(* CoDeSys 2.3.6.0 project: KOKEV_G53RT_8.pro *)
(* Libraries: STANDARD.LIB 5.6.98 12:03:02 *)

(* Task configuration *)
TASK Standard (PRIORITY := 0, INTERVAL := T#4ms);
	Nockenschaltwerk();
END_TASK

(* Global variable list: Globale_Variablen *)
VAR_GLOBAL
	E1  AT %IX0.0 : BOOL; (* Eingang 1 *)
	E2  AT %IX0.1 : BOOL; (* Eingang 2 *)
	E3  AT %IX0.2 : BOOL; (* Eingang 3 *)
	E4  AT %IX0.3 : BOOL; (* Eingang 4 *)
	E5  AT %IX0.4 : BOOL; (* Eingang 5 *)
	E6  AT %IX0.5 : BOOL; (* Eingang 6 *)
	E7  AT %IX0.6 : BOOL; (* Eingang 7 *)
	E8  AT %IX0.7 : BOOL; (* Eingang 8 *)

       E9  AT %IX1.0 : BOOL; (* Eingang 9 *)
	E10  AT %IX1.1 : BOOL; (* Eingang 10 *)
	E11  AT %IX1.2 : BOOL; (* Eingang 11 *)
	E12  AT %IX1.3 : BOOL; (* Eingang 12 *)
	E13  AT %IX1.4 : BOOL; (* Eingang 13 *)
	E14  AT %IX1.5 : BOOL; (* Eingang 14 *)
	_KS1_UmlRolleGeschl  AT %IX1.6 : BOOL; (* Speicher 1 ist geschloßen *)
	_KS2_UmlRolleGeschl  AT %IX1.7 : BOOL; (* Speicher 2 ist geschloßen *)

	E17  AT %IX2.0 : BOOL; (* Eingang 17 *)
	E18  AT %IX2.1 : BOOL; (* Eingang 18 *)
	E19  AT %IX2.2 : BOOL; (* Eingang 19 *)
	E20  AT %IX2.3 : BOOL; (* Eingang 20 *)
	E21  AT %IX2.4 : BOOL; (* Eingang 21 *)
	E22  AT %IX2.5 : BOOL; (* Eingang 22 *)
	E23  AT %IX2.6 : BOOL; (* Eingang 23 *)
	E24  AT %IX2.7 : BOOL; (* Eingang 24 *)

	T_Quitt_NA  AT %IX3.0 : BOOL; (* Eingang 9 *)
	T_Qiutt_Stoerung  AT %IX3.1 : BOOL; (* Eingang 10 *)
	T_Hand  AT %IX3.2 : BOOL; (* Eingang 11 *)
	T_Auto  AT %IX3.3 : BOOL; (* Eingang 12 *)
	T_Visu  AT %IX3.4 : BOOL; (* Eingang 13 *)
	T_KammBild  AT %IX3.5 : BOOL; (* Eingang 14 *)
	T_Start  AT %IX3.6 : BOOL; (* Eingang 15 *)
	T_Stop  AT %IX3.7 : BOOL; (* Eingang 16 *)

	ET9   AT %IX4.0 : BOOL; (* Eingang 17 *)
	ET10  AT %IX4.1 : BOOL; (* Eingang 18 *)
	ET11  AT %IX4.2 : BOOL; (* Eingang 19 *)
	ET12  AT %IX4.3 : BOOL; (* Eingang 20 *)
	ET13  AT %IX4.4 : BOOL; (* Eingang 21 *)
	ET14  AT %IX4.5 : BOOL; (* Eingang 22 *)
	T_KettenAnfang  AT %IX4.6 : BOOL; (* Eingang 23 *)
	ET16  AT %IX4.7 : BOOL; (* Eingang 24 *)


	IA_Pos_KS1_Input  AT%IW8:INT;	 	(*Speicher 1 Füllstand analoger Eingang*)
	IA_Pos_KS2_Input	AT%IW12:INT;   	(*Speicher 2 Füllstand analoger Eingang*)
	VW_Act_Pos_KS1: INT;					(*Aktueller Füllstand Kettenspeicher 1 skaliert*)
	VW_Act_Pos_KS2:INT;					(*Aktueller Füllstand Kettenspeicher 2 skaliert*)
	IA_EW3	AT%IW12:INT; 				(*Analogeingang 3*)
	IA_EW4  	AT%IW16:INT; 				(*Analogeingang 4*)
	IC_SSI_DG_Input  AT %ID20:UDINT;	(* Drehgeber *)
	My_IC_SSI_DG_Input:UDINT;

	_PneumPressEin  AT %QX0.0 : BOOL; (* Ventil Pneumatik  *)
	A2  AT %QX0.1 : BOOL; (* Ausgang 2 *)
	A3  AT %QX0.2 : BOOL; (* Ausgang 3 *)
	A4  AT %QX0.3 : BOOL; (* Ausgang 4 *)
	A5  AT %QX0.4 : BOOL; (* Ausgang 5 *)
	A6  AT %QX0.5 : BOOL; (* Ausgang 6 *)
	A7  AT %QX0.6 : BOOL; (* Ausgang 7 *)
	A8  AT %QX0.7 : BOOL; (* Ausgang 8 *)

	Q_KS2_EnOutput  AT %QX1.0 : BOOL; (* Ausgang 9 *)
	A10  AT %QX1.1 : BOOL; (* Ausgang 10 *)
	A11  AT %QX1.2 : BOOL; (* Ausgang 11 *)
	A12  AT %QX1.3 : BOOL; (* Ausgang 12 *)
	A13  AT %QX1.4 : BOOL; (* Ausgang 13 *)
	A14  AT %QX1.5 : BOOL; (* Ausgang 14 *)
	A15  AT %QX1.6 : BOOL; (* Ausgang 15 *)
	A16  AT %QX1.7 : BOOL; (* Ausgang 16 *)

	H_Quitt_NA  AT %QX2.0 : BOOL; (* Ausgang 1 *)
	H_Quitt_Stoerung  AT %QX2.1 : BOOL; (* Ausgang 2 *)
	H_Hand  AT %QX2.2 : BOOL; (* Ausgang 3 *)
	H_Auto  AT %QX2.3 : BOOL; (* Ausgang 4 *)
	H_Visu  AT %QX2.4 : BOOL; (* Ausgang 5 *)
	H_KammBild  AT %QX2.5 : BOOL; (* Ausgang 6 *)
	H_Start  AT %QX2.6 : BOOL; (* Ausgang 7 *)
	H_Stop  AT %QX2.7 : BOOL; (* Ausgang 8 *)

	AT9  AT %QX3.0 : BOOL; (* Ausgang 9 *)
	AT10  AT %QX3.1 : BOOL; (* Ausgang 10 *)
	AT11  AT %QX3.2 : BOOL; (* Ausgang 11 *)
	AT12  AT %QX3.3 : BOOL; (* Ausgang 12 *)
	AT13  AT %QX3.4 : BOOL; (* Ausgang 13 *)
	AT14  AT %QX3.5 : BOOL; (* Ausgang 14 *)
	H_KettenAnfang  AT %QX3.6 : BOOL; (* Ausgang 15 *)
	AT16  AT %QX3.7 : BOOL; (* Ausgang 16 *)


	QA_Sollw_Mot1   AT%QW4:WORD; (*Ausgangswort 1*)
	QA_Sollw_Mot2   AT%QW8:WORD; (*Ausgangswort 2*)

	KettenTypen			AT%QW100:ARRAY [1..10,0..10] OF INT ;	(* Es können maximal 10 Kettentypen definiert und remanent gespeichert werden *)
	AKT_KettenTyp		AT%QW420:INT;								(* Nummer des gültigen Kettentyps ( 1-10)   *)
	Speicher_Reg: ARRAY[0..500] OF WORD;							(* Speicherregister für Glieder es werden maximal 500 Glieder beobachtet *)
	Ketten_Reg: ARRAY[0..220] OF WORD;								(* Kettenregister für dien Aktuellen Kettentyp *)
	Z_AKT_KettenTyp_Max:INT;											(* Länge des Aktuellen Kettentyps *)
	Zeiger_Speicher_Trennstelle: INT;									(* Zeiger für die Glieder in der Anlage zeigt auf das Glied unter der Trennstelle *)
	Zeiger_Kette_Trennstelle:INT;										(* Zeiger für die Glieder der Kette zeigt auf das Glied unter der Trennstelle*)
	Zeiger_Loeschen: INT;												(* Zeiger zum Löschen der Register beim Überlauf *)
	M1:BOOL;

	CTU1: CTU;
END_VAR

(* Data type *)
TYPE DriveControl :
STRUCT
	ManOn: BOOL := FALSE; (* Visu -> SPS: Antrieb ein (nur bei FU-Antrieben) *)
	ManOff: BOOL := FALSE; (* Visu -> SPS: Antrieb aus (nur bei FU-Antrieben) *)
	ManFwd: BOOL := FALSE; (* Visu -> SPS: Antrieb im Handbetrieb langsam vorwärts *)
	ManBwd: BOOL := FALSE; (* Visu -> SPS: Antrieb im Handbetrieb langsam rückwärts *)
	TeilungVor: BOOL := FALSE; (* Visu -> SPS: Kette um eine Teilung vor (nur bei Servo-Antrieben) *)
	TeilungZur: BOOL := FALSE; (* Visu -> SPS: Kette um eine Teilung zurück (nur bei Servo-Antrieben) *)
	EnManCtrl: BOOL := FALSE; (* SPS -> Visu: Freigabe manuelle Steuerung *)
	ActOn: BOOL := FALSE; (* SPS -> Visu: Antrieb eingeschaltet *)
	ActOff: BOOL := FALSE; (* SPS -> Visu: Antrieb ausgeschaltet *)
	Error: BOOL := FALSE; (* SPS -> Visu: Störung Antrieb *)
END_STRUCT
END_TYPE

(* Data type *)
TYPE KettenTyp :
STRUCT
	PF: ARRAY [0..19] OF UDINT := 0,410,819,1229,1638,2048,2458,2867,3277,3686,4049,4506,4915,5328,5734,6144,6554,6963,7373,7782;

END_STRUCT
END_TYPE

(* Data type *)
TYPE KS_Control :
STRUCT
	EnInput: BOOL := FALSE; (* Freigabe Befüllen *)
	EnOutput: BOOL := FALSE; (* Freigabe Entleeren *)
	ActState: INT := 0; (* aktueller zustand für Visu *)
END_STRUCT
END_TYPE

(* Data type *)
TYPE MotorControl :
STRUCT
	ManOn: BOOL := FALSE; (* Visu -> SPS: Antrieb im Handbetrieb ein *)
	ManOff: BOOL := FALSE; (* Visu -> SPS: Antrieb im Handbetrieb aus *)
	EnManCtrl: BOOL := FALSE; (* SPS -> Visu: Freigabe manuelle Steuerung *)
	ActOn: BOOL := FALSE; (* SPS -> Visu: Antrieb eingeschaltet *)
	ActOff: BOOL := FALSE; (* SPS -> Visu: Antrieb ausgeschaltet *)
	Error: BOOL := FALSE; (* SPS -> Visu: Störung Antrieb *)
END_STRUCT
END_TYPE

(* Data type *)
TYPE PneumControl :
STRUCT
	SetOn: BOOL := FALSE; (* Visu -> SPS: Arbeitsstellung anfahren *)
	SetOff: BOOL := FALSE; (* Visu -> SPS: Grundstellung anfahren *)
	EnSet: BOOL := FALSE; (* SPS -> Visu: Freigabe manuell Steuerung *)
	ActOn: BOOL := FALSE; (* SPS -> Visu: Zylinder in Arbeitsstellung *)
	ActOff: BOOL := FALSE; (* SPS -> Visu: Zylinder in Grundstellung *)
	Error: BOOL := FALSE; (* SPS -> Visu: Störung Zylinder oder Endschalter *)
END_STRUCT
END_TYPE

(* Data type *)
TYPE PosControl :
STRUCT
	PosSet: INT := 0; (* Positionssollwert [mm] *)
	ActPos: INT := 0; (* Positionsistwert [mm] *)
	PosLimitLo: INT := 0; (* unterer Grenzwert Sollposition [mm] *)
	PosLimitHi: INT := 0; (* oberer Grenzwert Sollposition [mm] *)
	StartPos: BOOL := FALSE; (* Visu -> SPS: Positionierung starten *)
	StoppPos: BOOL := FALSE; (* Visu -> SPS: Positionierung abbrechen *)
	ManPosUp: BOOL := FALSE; (* Visu -> SPS: Handbetrieb Positon erhöhen *)
	ManPosDn: BOOL := FALSE; (* Visu -> SPS: Handbetrieb Positon verringern *)
	EnPosSet: BOOL := FALSE; (* SPS -> Visu: Freigabe Sollwerteingabe *)
	EnManPos: BOOL := FALSE; (* SPS -> Visu: Freigabe manuelle Positionierung *)
	ActOn: BOOL := FALSE; (* SPS -> Visu: Antrieb eingeschaltet *)
	ActOff: BOOL := FALSE; (* SPS -> Visu: Antrieb ausgeschaltet *)
	Error: BOOL := FALSE; (* SPS -> Visu: Störung Antrieb *)
END_STRUCT
END_TYPE

(* Data type *)
TYPE StationControl :
STRUCT
	StepCounter: INT; (* SPS -> Visu: Schrittzähler *)
	SingleStep: BOOL := FALSE; (* Visu -> SPS: Einzelschritt weiterschalten *)
	SingleCycle: BOOL := FALSE; (* Visu -> SPS: Einzelzyklus ausführen *)
	StartCycle: BOOL := FALSE; (* Zyklus im Auto-Betrieb starten *)
	ManInit: BOOL := FALSE; (* Visu -> SPS: Grundstellung anfahren *)
	AutoInit: BOOL := FALSE; (* Grundstellung im Auto-Betrieb anfahren *)
	SetFinished: BOOL := FALSE; (* Visu -> SPS: Fertigmeldung setzen *)
	WaitPos: BOOL := FALSE; (* Station in Warteposition für Stopp *)
	EnSemiAutoCtrl: BOOL := FALSE; (* SPS -> Visu: Steuerung Halbautomatikbetrieb freigeben; Freigabe für SingleStep, SingleCycle, InitPos und SetFinished *)
	InitPos: BOOL := FALSE; (* Station in Grundstellung *)
	Finished: BOOL := FALSE; (* Station fertig *)
	ErrorInitPos: BOOL := FALSE; (* Störung Grundstellung nicht erreicht *)
	ErrorCycleTime: BOOL := FALSE; (* Störung Zeitüberschreitung Zyklus *)
	ActState: INT := 0; (* SPS -> Visu: Zustand der Station: 0 = Störung, 1 = bereit, 2 = aktiv *)
END_STRUCT
END_TYPE

(* POU Nockenschaltwerk, ST *)
PROGRAM Nockenschaltwerk
VAR
	Zeiger :INT:=0;
	Nocke:BOOL:=FALSE;
	Zaeler:WORD;
	Skal_IC_SSI_DG_Input: DINT;
	Skal_IC_SSI_DG_Input_Alt:DINT;
	Skal_IC_SSI_DG_Input_Delta:DINT;
	CTU2:WORD;
END_VAR
(*  Miroslav Knezevic TCM 19.03.07  *)
(*  Das Nockenschaltwerk liefert 20 Impulse bei einer Umdrehung des SSI Drehgebers *)
(* Voller Kreis = 8192 Inkremente,  1 Impuls= 20 Inkremente *)



Skal_IC_SSI_DG_Input:=IC_SSI_DG_Input* 20 / 256;
Skal_IC_SSI_DG_Input_Delta:=Skal_IC_SSI_DG_Input - Skal_IC_SSI_DG_Input_Alt;

IF Skal_IC_SSI_DG_Input_Delta<-5 THEN
	Skal_IC_SSI_DG_Input_Delta:=1;
END_IF

IF Skal_IC_SSI_DG_Input_Delta>5 THEN
	Skal_IC_SSI_DG_Input_Delta:=-1;
END_IF

Zeiger_Speicher_Trennstelle:=DINT_TO_INT(Zeiger_Speicher_Trennstelle+Skal_IC_SSI_DG_Input_Delta);
IF Zeiger_Speicher_Trennstelle>500 THEN
	Zeiger_Speicher_Trennstelle:=1;
END_IF
IF Zeiger_Speicher_Trennstelle<1 THEN
	Zeiger_Speicher_Trennstelle:=500;
END_IF

CTU1(
	CU:=M1 ,
	RESET:= ,
	PV:=500 ,
	Q=> ,
	CV=> );

CTU2:=CTU1.CV;


Zeiger_Kette_Trennstelle:=DINT_TO_INT(Zeiger_Kette_Trennstelle+Skal_IC_SSI_DG_Input_Delta);
IF Zeiger_Kette_Trennstelle>Z_AKT_KettenTyp_Max THEN
	Zeiger_Kette_Trennstelle:=1;
END_IF

IF Zeiger_Kette_Trennstelle<1 THEN
	Zeiger_Kette_Trennstelle:=Z_AKT_KettenTyp_Max;
END_IF

IF ABS(Skal_IC_SSI_DG_Input_Delta)>1 THEN
		M1:=TRUE;

END_IF

Skal_IC_SSI_DG_Input_Alt:=Skal_IC_SSI_DG_Input;
END_PROGRAM

(* POU Funktionsbausteine/_ASM_FU_SOLLW, ST *)
FUNCTION_BLOCK _ASM_FU_SOLLW
VAR_INPUT
	SollW: INT;
	IstW:INT;
	P:INT;
	Pos_Fenster:INT;
END_VAR
VAR_OUTPUT
	SollwReg:INT;
	Vor_Rueck:BOOL;
	Pos_Erreicht:BOOL;
END_VAR
VAR
END_VAR
IF SollW>=IstW THEN
		SollwReg := ( SollW-IstW) *P;
		Vor_Rueck := TRUE;
ELSE
		SollwReg := ( IstW-SollW) *P;
		Vor_Rueck := FALSE;
END_IF

IF ABS( SollW-IstW)<Pos_Fenster THEN
		Pos_Erreicht := TRUE;
ELSE
		Pos_Erreicht := FALSE;
END_IF
END_FUNCTION_BLOCK

(* POU Funktionsbausteine/ClearTestArrays, ST *)
FUNCTION_BLOCK ClearTestArrays
VAR CONSTANT
	ClearArray: ARRAY[0..7] OF INT := 8(0);
END_VAR
VAR_INPUT
	enable: BOOL := FALSE; (* Freigabe *)
END_VAR
VAR_IN_OUT
	Gelenk_I: ARRAY[0..7] OF INT;
	Gelenk_A: ARRAY[0..7] OF INT;
	Vollstaendigkeit: ARRAY[0..7] OF INT;
	Nietung: ARRAY[0..7] OF INT;
	ZZP: ARRAY[0..7] OF INT;
	Huelse: ARRAY[0..7] OF INT;
END_VAR
IF enable THEN

	Gelenk_I			:= ClearArray;
	Gelenk_A			:= ClearArray;
	Vollstaendigkeit	:= ClearArray;
	Nietung			:= ClearArray;
	ZZP				:= ClearArray;
	Huelse			:= ClearArray;

END_IF;
END_FUNCTION_BLOCK

(* POU Funktionsbausteine/ClockDivide, ST *)
FUNCTION_BLOCK ClockDivide
VAR
	clock_old: BOOL;
	counter: INT;
END_VAR
VAR_INPUT
	clock_in: BOOL; (* clock input *)
	n: INT; (* divider *)
END_VAR
VAR_OUTPUT
	clock_out: BOOL;
END_VAR
IF n < 1 THEN n := 1;
END_IF;

IF NOT clock_old AND clock_in AND counter <= n THEN
	counter := counter + 1;
END_IF;

IF counter >= n THEN
	clock_out  := NOT clock_out;
	counter := 0;
END_IF;

clock_old := clock_in;
END_FUNCTION_BLOCK

(* POU Funktionsbausteine/ErrMove, ST *)
FUNCTION_BLOCK ErrMove
VAR
	i: INT;
	n: INT;
END_VAR
VAR_INPUT
	ErrArray: ARRAY[0..511] OF BOOL;
END_VAR
VAR_OUTPUT
	ErrWordArray: ARRAY[0..31] OF WORD;
END_VAR
FOR i := 0 TO 31 DO
	n := i * 16;
	ErrWordArray[i].0 := ErrArray[n];
	ErrWordArray[i].1 := ErrArray[n+1];
	ErrWordArray[i].2 := ErrArray[n+2];
	ErrWordArray[i].3 := ErrArray[n+3];
	ErrWordArray[i].4 := ErrArray[n+4];
	ErrWordArray[i].5 := ErrArray[n+5];
	ErrWordArray[i].6 := ErrArray[n+6];
	ErrWordArray[i].7 := ErrArray[n+7];
	ErrWordArray[i].8 := ErrArray[n+8];
	ErrWordArray[i].9 := ErrArray[n+9];
	ErrWordArray[i].10 := ErrArray[n+10];
	ErrWordArray[i].11 := ErrArray[n+11];
	ErrWordArray[i].12 := ErrArray[n+12];
	ErrWordArray[i].13 := ErrArray[n+13];
	ErrWordArray[i].14 := ErrArray[n+14];
	ErrWordArray[i].15 := ErrArray[n+15];
END_FOR;
END_FUNCTION_BLOCK

(* POU Funktionen/IntScale, ST *)
FUNCTION IntScale : INT
VAR_INPUT
	Int_In: INT; (* Eingangsvariable *)
	Real_Scale: REAL; (* Skalierfaktor *)
	Int_Zero: INT; (* Nullpunkt *)
END_VAR
IntScale := REAL_TO_INT ( ( INT_TO_REAL ( Int_In ) * Real_Scale ) ) + Int_Zero;
END_FUNCTION

(* POU Funktionsbausteine/Kettenregister, ST *)
FUNCTION_BLOCK Kettenregister
VAR_INPUT

END_VAR
VAR_OUTPUT
END_VAR
VAR

	AKT_KettenTyp_Alt: INT;

END_VAR
IF AKT_KettenTyp<>AKT_KettenTyp_Alt THEN
	Z_AKT_KettenTyp_Max:=KettenTypen[AKT_KettenTyp,0]-1;
	Ketten_Reg[KettenTypen[AKT_KettenTyp,1]*2]:=KettenTypen[AKT_KettenTyp,2];
	Ketten_Reg[KettenTypen[AKT_KettenTyp,3]*2]:=KettenTypen[AKT_KettenTyp,4];
	Ketten_Reg[KettenTypen[AKT_KettenTyp,5]*2]:=KettenTypen[AKT_KettenTyp,6];
	Ketten_Reg[KettenTypen[AKT_KettenTyp,7]*2]:=KettenTypen[AKT_KettenTyp,8];
	Ketten_Reg[KettenTypen[AKT_KettenTyp,10]*2]:=KettenTypen[AKT_KettenTyp,10];
END_IF
AKT_KettenTyp_Alt:=AKT_KettenTyp;
END_FUNCTION_BLOCK

(* POU Funktionsbausteine/KS, ST *)
FUNCTION_BLOCK KS
VAR_INPUT
	URL_Geschlossen: BOOL; (* Umlenkrolle geschlossen *)
	SpannzylinderGespannt: BOOL; (* Spannzylinder Kettenspeicher gespannt *)
	ActPress: INT; (* Druck-Istwert Spannzylinder *)
	ActPos_ULR: INT; (* Positions-Istwert Umlenkrolle *)
	MinPress: INT; (* minimaler Druck Spannzylinder *)
	MaxPress: INT; (* maximaler Druck Spannzylinder *)
	MinPos_ULR: INT; (* minimale Position Umlenkrolle *)
	MaxPos_ULR: INT; (* maximale Position Umlenkrolle *)
	MaxKapazitaet: INT; (* maximale Kettenspeicher-Kapazität in Gliedern *)
	Gliederzahl_InTakt: INT; (* Gliederzahl für getaktetes Befüllen (0 = konstante Geschwindigkeit) *)
	Gliederzahl_OutTakt: INT; (* Gliederzahl für getaktete Entnahme (0 = konstante Geschwindigkeit) *)
END_VAR
VAR_OUTPUT
	En_Input: BOOL; (* Freigabe Befüllen *)
	En_Output: BOOL; (* Freigabe Entnahme *)
	ActState: INT; (* aktueller Zustand für Visu *)
END_VAR
VAR
	KS_ready: BOOL; (* Kettenspeicher bereit *)
	ActKapazitaet: INT; (* aktuelle Kettenspeicher-Kapazität in Gliedern *)
END_VAR
(* Kettenspeicher betriebsbereit *)

KS_ready := ActPress >= MinPress AND ActPress <= MaxPress AND URL_Geschlossen AND SpannzylinderGespannt;

(* Berechnung der aktuellen Kettenspeicher-Kapazität in Gliedern *)

(* ActKapazitaet := LIMIT (MinPos_ULR, MaxPos_ULR - ActPos_ULR, MaxPos_ULR) * MaxKapazitaet / ( MaxPos_ULR - MinPos_ULR ); *)
ActKapazitaet := ( 32767 - LIMIT (MinPos_ULR, ActPos_ULR, MaxPos_ULR) ) * MaxKapazitaet / ( MaxPos_ULR - MinPos_ULR );


(* Freigaben für Befüllen *)

IF Gliederzahl_InTakt = 0 THEN
	IF ActKapazitaet < ( MaxKapazitaet * 3 / 4 ) AND KS_ready THEN
		En_Input := TRUE;					(* Befüllung mit konstanter Geschwindigkeit: mindestens 25% Kapazität im Kettenspeicher frei *)
	END_IF;
	IF ActKapazitaet >= MaxKapazitaet OR NOT KS_ready THEN
		En_Input := FALSE;					(* Kettenspeicher voll *)
	END_IF;
ELSE
	En_Input := ActKapazitaet <= (MaxKapazitaet - Gliederzahl_InTakt) AND KS_ready;		(* getaktete Befüllung: mindestens 1 Stranglänge im Kettenspeicher frei *)
END_IF;


(* Freigaben für Entnahme *)

IF Gliederzahl_OutTakt = 0 THEN
	IF ActKapazitaet > MaxKapazitaet / 4 AND KS_ready THEN
		En_Output := TRUE;					(* Entnahme mit konstanter Geschwindigkeit: mindestens 25% Kapazität im Kettenspeicher belegt *)
	END_IF;
	IF ActKapazitaet <= 0 OR NOT KS_ready THEN
		En_Output := FALSE;					(* Kettenspeicher leer *)
	END_IF;
ELSE
	En_Output := ActKapazitaet >= Gliederzahl_OutTakt AND KS_ready;		(* getaktete Befüllung: mindestens 1 Stranglänge im Kettenspeicher belegt *)
END_IF;


(* Freigaben sperren wenn Kettenspeicher nicht bereit (offen oder entspannt oder Druck nicht OK *)

IF NOT KS_ready THEN
	En_Input := FALSE;
	En_Output := FALSE;
END_IF;

(* aktueller Zustand für Visu *)

IF KS_ready THEN
	ActState := 1;				(* bereit *)
ELSE
	ActState := 0;				(* Störung *)
END_IF;
END_FUNCTION_BLOCK

(* POU Funktionsbausteine/OutCtrlB, ST *)
FUNCTION_BLOCK OutCtrlB
VAR
	TO_Zyl: TON;
END_VAR
VAR_INPUT
	AutoSet: BOOL := FALSE; (* Ausgang im Automatikbetrieb einschalten *)
	AutoReset: BOOL := FALSE; (* Ausgang im Automatikbetrieb ausschalten *)
	AutoEnable: BOOL := FALSE; (* Ausgangsfreigabe im Auto-Betrieb *)
	ManEnable: BOOL := FALSE; (* Ausgangsfreigabe im Handbetrieb *)
	INI_Home: BOOL := FALSE; (* Initiator Grundstellung *)
	INI_End: BOOL := FALSE; (* Initiator Arbeitsstellung *)
	HoldHome: BOOL := FALSE; (* Ventil in Grundstellung bestromen *)
	HoldEnd: BOOL := FALSE; (* Ventil in Arbeitsstellung bestromen *)
	ResetError: BOOL := FALSE; (* Störung rücksetzen *)
	ManualMode: BOOL := FALSE; (* Betriebsart Hand *)
	Timeout: TIME; (* Zeitüberwachung *)
	clock: BOOL := FALSE; (* Takt für Störung *)
END_VAR
VAR_OUTPUT
	OutEnd: BOOL; (* Ausgang Endstellung für bistabiles Magnetventil *)
	OutHome: BOOL; (* Ausgang Endstellung für bistabiles Magnetventil *)
	EnManControl: BOOL; (* Freigabe Visu-Steuerung Handbetrieb *)
	ActEnd: BOOL; (* aktueller Zustand eingeschaltet *)
	ActHome: BOOL; (* aktueller Zustand ausgeschaltet *)
	VisuErrorState: BOOL; (* Störmeldung für Visu *)
	Error: BOOL; (* Störung Pneumatikzylinder oder Endschalter *)
END_VAR
VAR_IN_OUT
	ManSet: BOOL; (* Ausgang im Manuellbetrieb einschalten *)
	ManReset: BOOL; (* Ausgang im Manuellbetrieb ausschalten *)
END_VAR
IF  ( AutoSet AND AutoEnable ) OR ( ManSet AND ManEnable ) THEN							(* Ausgang Arbeitsstellung einschalten *)
	OutEnd := TRUE;
	OutHome := FALSE;
END_IF;

IF ( NOT AutoEnable AND NOT ManEnable ) OR ( INI_End AND NOT HoldEnd ) OR Error THEN
	OutEnd := FALSE;												(* Ausgang Arbeitsstellung ausschalten *)
END_IF;

IF ( AutoReset AND AutoEnable ) OR ( ManReset AND ManEnable ) THEN						(* Ausgang Grundstellung einschalten *)
	OutHome := TRUE;
	OutEnd := FALSE;
END_IF;

IF ( NOT AutoEnable AND NOT ManEnable ) OR ( INI_Home AND NOT HoldHome ) OR Error THEN
	OutHome := FALSE;												(* Ausgang Grundstellung ausschalten *)
END_IF;


(* Aktueller Zustand *)

ActEnd := INI_End AND NOT INI_Home;
ActHome := INI_Home AND NOT INI_End;

(* Störung Pneumatikzylinder *)

TO_Zyl ( IN := ( ( OutEnd AND ( INI_Home OR NOT INI_End ) ) OR ( OutHome AND ( INI_End OR NOT INI_Home ) ) OR ( INI_Home AND INI_End )) ,
	 PT := Timeout );
IF TO_Zyl.Q  THEN
	Error := TRUE;
ELSIF ResetError THEN
	Error := FALSE;
END_IF;

(* Störungsmeldung für Visu aktivieren *)

VisuErrorState := Error OR ( clock AND ( ( AutoSet AND NOT INI_End ) OR ( AutoReset AND NOT INI_Home ) ) );

(* Freigabe Visu-Steuerbuttons im Handbetrieb *)

EnManControl := ManualMode AND ManEnable AND NOT Error;

(* Visu-Steuerbuttons für Handbetrieb rücksetzen *)

ManSet := FALSE;
ManReset := FALSE;
END_FUNCTION_BLOCK

(* POU Funktionsbausteine/OutCtrlKS, ST *)
FUNCTION_BLOCK OutCtrlKS
VAR
	AutoOn: BOOL := FALSE; (* Ausgang im Auto-Betrieb einschalten *)
	ManOn: BOOL := FALSE; (* Ausgang im Manuell-Betrieb einschalten *)
	TO_Zyl: TON;
END_VAR
VAR_INPUT
	AutoSet: BOOL := FALSE; (* Ausgang im Automatikbetrieb einschalten *)
	AutoReset: BOOL := FALSE; (* Ausgang im Automatikbetrieb ausschalten *)
	AutoEnable: BOOL := FALSE; (* Ausgangsfreigabe für Auto-Betrieb *)
	ManEnable: BOOL := FALSE; (* Ausgangsfreigabe für Handbetrieb *)
	ErrEnable: BOOL := FALSE; (* Freigabe Fehlerauswertung *)
	INI_Home: BOOL := FALSE; (* Initiator Grundstellung *)
	INI_End: BOOL := FALSE; (* Initiator Arbeitsstellung *)
	ManualMode: BOOL; (* Betriebsart Hand *)
	Timeout: TIME; (* Zeitüberwachung *)
	ResetError: BOOL; (* Störung rücksetzen *)
	clock: BOOL := FALSE; (* Takt für Störung *)
END_VAR
VAR_OUTPUT
	Output: BOOL; (* Ausgang für monostabiles Magnetventil *)
	EnManControl: BOOL; (* Freigabe Handsteuerung für Visu *)
	ActEnd: BOOL; (* aktueller Zustand eingeschaltet *)
	ActHome: BOOL; (* aktueller Zustand ausgeschaltet *)
	VisuErrorState: BOOL; (* Fehlermeldung aktivieren *)
	Error: BOOL; (* Störung Pneumatikzylinder oder Endschalter *)
END_VAR
VAR_IN_OUT
	ManSet: BOOL; (* Ausgang im Manuellbetrieb einschalten *)
	ManReset: BOOL; (* Ausgang im Manuellbetrieb ausschalten *)
END_VAR
IF AutoEnable AND NOT ManEnable AND AutoSet AND NOT Error THEN
	AutoOn := TRUE;									(* Ausgang im Auto-Betrieb einschalten *)
END_IF;

IF ManEnable AND ManSet AND NOT Error THEN
	ManOn := TRUE;									(* Ausgang im Handbetrieb einschalten *)
	ManSet := FALSE;
END_IF;

IF NOT AutoEnable OR ( AutoEnable AND ManEnable AND ManReset ) OR AutoReset OR Error THEN
	AutoOn := FALSE;									(* Ausgang im Auto-Betrieb ausschalten *)
END_IF;

IF NOT ManEnable OR ManReset OR Error THEN
	ManOn := FALSE;									(* Ausgang im Handbetrieb ausschalten *)
	ManReset := FALSE;
END_IF;

Output := AutoOn OR ManOn;							(* Ausgang zuweisen *)

(* Aktueller Zustand *)

ActEnd := INI_End AND NOT INI_Home;
ActHome := INI_Home AND NOT INI_End;

(* Störung Pneumatikzylinder *)

TO_Zyl ( IN := ( ( Output AND ( INI_Home OR NOT INI_End ) ) OR ( NOT Output AND ( INI_End OR NOT INI_Home ) ) ) , PT := Timeout );
IF ErrEnable AND (TO_Zyl.Q OR ( INI_Home AND INI_End )) THEN
	Error := TRUE;
ELSIF ResetError THEN
	Error := FALSE;
END_IF;


(* Störungsmeldung für Visu aktivieren *)

VisuErrorState := Error OR ( clock AND ( ( AutoSet AND NOT INI_End ) OR ( AutoReset AND NOT INI_Home ) ) );


(* Freigabe Visu-Steuerbuttons im Handbetrieb *)

EnManControl := ManualMode AND NOT Error;
END_FUNCTION_BLOCK

(* POU Funktionsbausteine/OutCtrlM, ST *)
FUNCTION_BLOCK OutCtrlM
VAR
	AutoOn: BOOL := FALSE; (* Ausgang im Auto-Betrieb einschalten *)
	ManOn: BOOL := FALSE; (* Ausgang im Manuell-Betrieb einschalten *)
	TO_Zyl: TON;
END_VAR
VAR_INPUT
	AutoSet: BOOL := FALSE; (* Ausgang im Automatikbetrieb einschalten *)
	AutoReset: BOOL := FALSE; (* Ausgang im Automatikbetrieb ausschalten *)
	AutoEnable: BOOL := FALSE; (* Ausgangsfreigabe für Auto-Betrieb *)
	ManEnable: BOOL := FALSE; (* Ausgangsfreigabe für Handbetrieb *)
	ErrEnable: BOOL := FALSE; (* Freigabe Fehlerauswertung *)
	INI_Home: BOOL := FALSE; (* Initiator Grundstellung *)
	INI_End: BOOL := FALSE; (* Initiator Arbeitsstellung *)
	ManualMode: BOOL; (* Betriebsart Hand *)
	Timeout: TIME; (* Zeitüberwachung *)
	ResetError: BOOL; (* Störung rücksetzen *)
	clock: BOOL := FALSE; (* Takt für Störung *)
END_VAR
VAR_OUTPUT
	Output: BOOL; (* Ausgang für monostabiles Magnetventil *)
	EnManControl: BOOL; (* Freigabe Handsteuerung für Visu *)
	ActEnd: BOOL; (* aktueller Zustand eingeschaltet *)
	ActHome: BOOL; (* aktueller Zustand ausgeschaltet *)
	VisuErrorState: BOOL; (* Fehlermeldung aktivieren *)
	Error: BOOL; (* Störung Pneumatikzylinder oder Endschalter *)
END_VAR
VAR_IN_OUT
	ManSet: BOOL; (* Ausgang im Manuellbetrieb einschalten *)
	ManReset: BOOL; (* Ausgang im Manuellbetrieb ausschalten *)
END_VAR
IF AutoEnable  AND AutoSet AND NOT Error THEN
	AutoOn := TRUE;									(* Ausgang im Auto-Betrieb einschalten *)
END_IF;

IF ManEnable AND ManSet AND NOT Error THEN
	ManOn := TRUE;									(* Ausgang im Handbetrieb einschalten *)
	ManSet := FALSE;
END_IF;

IF NOT AutoEnable OR ( AutoEnable AND ManEnable AND ManReset ) OR AutoReset OR Error THEN
	AutoOn := FALSE;									(* Ausgang im Auto-Betrieb ausschalten *)
END_IF;

IF NOT ManEnable OR ManReset OR Error THEN
	ManOn := FALSE;									(* Ausgang im Handbetrieb ausschalten *)
	ManReset := FALSE;
END_IF;

Output := AutoOn OR ManOn;							(* Ausgang zuweisen *)

(* Aktueller Zustand *)

ActEnd := INI_End AND NOT INI_Home;
ActHome := INI_Home AND NOT INI_End;

(* Störung Pneumatikzylinder *)

TO_Zyl ( IN := ( ( Output AND ( INI_Home OR NOT INI_End ) ) OR ( NOT Output AND ( INI_End OR NOT INI_Home ) ) ) , PT := Timeout );
IF ErrEnable AND (TO_Zyl.Q OR ( INI_Home AND INI_End )) THEN
	Error := TRUE;
ELSIF ResetError THEN
	Error := FALSE;
END_IF;


(* Störungsmeldung für Visu aktivieren *)

VisuErrorState := Error OR ( clock AND ( ( AutoSet AND NOT INI_End ) OR ( AutoReset AND NOT INI_Home ) ) );


(* Freigabe Visu-Steuerbuttons im Handbetrieb *)

EnManControl := ManualMode AND NOT Error;
END_FUNCTION_BLOCK

(* POU Funktionsbausteine/ServoKette, FBD *)
FUNCTION_BLOCK ServoKette
VAR

	TOF_RFR: TOF; (* Ausschaltverzögerung Reglerfreigabe *)
END_VAR
VAR_INPUT
	AutoStartPos: BOOL := FALSE; (* Automatikbetrieb Positionierung starten *)
	ManFwd: BOOL := FALSE; (* Handbetrieb vorwärts *)
	ManBwd: BOOL := FALSE; (* Handbetrieb rückwärts *)
	ManualMode: BOOL := FALSE; (* Betriebsart Manuell *)
	NotAusOK: BOOL := FALSE; (* Not-Aus OK *)
	DriveError: BOOL := FALSE; (* Antriebsstörung *)
	Servo_Ready: BOOL := FALSE; (* Antrieb bereit *)
	RefError: BOOL := FALSE; (* Störung Referenzierung *)
	PosError: BOOL := FALSE; (* Störung Positionierung *)
	ResetError: BOOL := FALSE; (* Störung rücksetzen *)
	Clock: BOOL := FALSE; (* Takt für Fehler *)
END_VAR
VAR_OUTPUT
	Servo_RFR: BOOL := FALSE; (* Servoumrichter Reglerfreigabe *)
	Servo_CINH: BOOL := FALSE; (* Servoumrichter Reglersperre über CAN-Bus *)
	ServoManFwd: BOOL := FALSE; (* Servoantrieb manuell vorwärts *)
	ServoManBwd: BOOL := FALSE; (* Servoantrieb manuell rückwärts *)
	ServoStartPos: BOOL := FALSE; (* Servoantrieb Positionierung starten *)
	ServoTripReset: BOOL := FALSE; (* Servoumrichter Störung rücksetzen *)
	ServoResetError: BOOL := FALSE; (* Servoumrichter Störung Ref/Pos zurücksetzen *)
	EnManCtrl: BOOL := FALSE; (* Freigabe manuelle Steuerung *)
	Visu_DriveOn: BOOL := FALSE; (* Visu: Antrieb eingeschaltet *)
	Visu_DriveOff: BOOL := FALSE; (* Visu: Antrieb ausgeschaltet *)
	Visu_Error: BOOL := FALSE; (* Visu: Störung Antrieb *)
	Error: BOOL := FALSE; (* Sammelstörung Antrieb *)
END_VAR
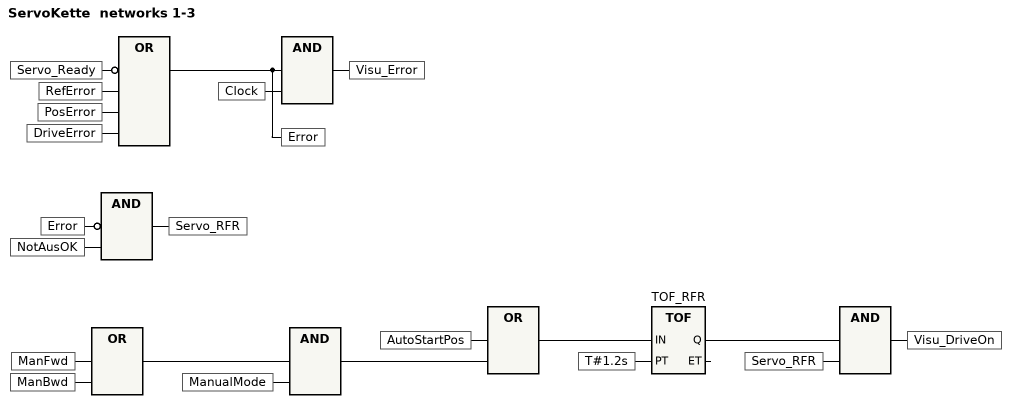
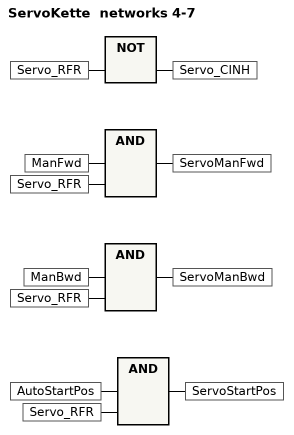
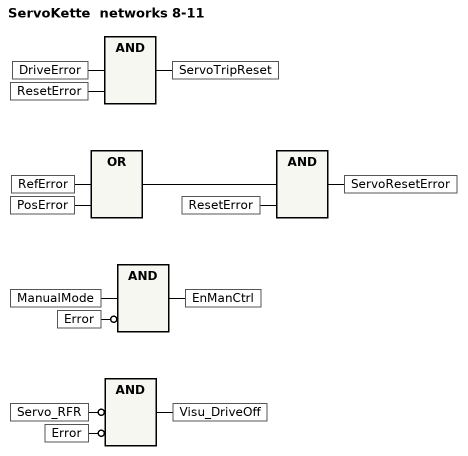
_FBD_ (* Function Block Diagram *)
NETWORK 1 (* Störung Antrieb *)
	AND(<OR(NOT Servo_Ready, RefError, PosError, DriveError) => Error>, Clock) => Visu_Error
NETWORK 2 (* Ausgang Reglerfreigabe *)
	AND(NOT Error, NotAusOK) => Servo_RFR
NETWORK 3 (* Antrieb ein für Visu *)
	AND(TOF_RFR:TOF(IN: OR(AutoStartPos, AND(OR(ManFwd, ManBwd), ManualMode)), PT: T#1.2s), Servo_RFR) => Visu_DriveOn
NETWORK 4 (* Ausgang Reglersperre *)
	NOT Servo_RFR => Servo_CINH
NETWORK 5 (* Ausgang manuell vorwärts *)
	AND(ManFwd, Servo_RFR) => ServoManFwd
NETWORK 6 (* Ausgang manuell rückwärts *)
	AND(ManBwd, Servo_RFR) => ServoManBwd
NETWORK 7 (* Ausgang Auto-Positionierung starten *)
	AND(AutoStartPos, Servo_RFR) => ServoStartPos
NETWORK 8 (* Ausgang Trip Reset *)
	AND(DriveError, ResetError) => ServoTripReset
NETWORK 9 (* Ausgang Störung Ref/Pos rücksetzen *)
	AND(OR(RefError, PosError), ResetError) => ServoResetError
NETWORK 10 (* Freigabe für Visu-Steuerbuttons Handbetrieb *)
	AND(ManualMode, NOT Error) => EnManCtrl
NETWORK 11 (* Visu: Antrieb ausgeschaltet *)
	AND(NOT Servo_RFR, NOT Error) => Visu_DriveOff
_END_FBD_
(* the same logic as Structured Text *)
(* Network 1: Störung Antrieb *)
Error := NOT Servo_Ready OR RefError OR PosError OR DriveError;
Visu_Error := Error AND Clock;
(* Network 2: Ausgang Reglerfreigabe *)
Servo_RFR := NOT Error AND NotAusOK;
(* Network 3: Antrieb ein für Visu *)
TOF_RFR(IN := AutoStartPos OR ((ManFwd OR ManBwd) AND ManualMode), PT := T#1.2s);
Visu_DriveOn := TOF_RFR.Q AND Servo_RFR;
(* Network 4: Ausgang Reglersperre *)
Servo_CINH := NOT Servo_RFR;
(* Network 5: Ausgang manuell vorwärts *)
ServoManFwd := ManFwd AND Servo_RFR;
(* Network 6: Ausgang manuell rückwärts *)
ServoManBwd := ManBwd AND Servo_RFR;
(* Network 7: Ausgang Auto-Positionierung starten *)
ServoStartPos := AutoStartPos AND Servo_RFR;
(* Network 8: Ausgang Trip Reset *)
ServoTripReset := DriveError AND ResetError;
(* Network 9: Ausgang Störung Ref/Pos rücksetzen *)
ServoResetError := (RefError OR PosError) AND ResetError;
(* Network 10: Freigabe für Visu-Steuerbuttons Handbetrieb *)
EnManCtrl := ManualMode AND NOT Error;
(* Network 11: Visu: Antrieb ausgeschaltet *)
Visu_DriveOff := NOT Servo_RFR AND NOT Error;
END_FUNCTION_BLOCK

(* POU Funktionen/State, ST *)
FUNCTION State : INT
VAR_INPUT
	error: BOOL := FALSE; (* Störung *)
	busy: BOOL := FALSE; (* Station aktiv *)
	finished: BOOL := FALSE; (* Station fertig *)
END_VAR
IF NOT error AND NOT busy THEN
	IF finished THEN
		State := 3;							(* Station fertig *)
	ELSE
		State := 1;							(* Station bereit *)
	END_IF;
ELSIF busy AND NOT error THEN
	State := 2;								(* Station aktiv *)
ELSE
	State := 0;								(* Störung *)
END_IF;
END_FUNCTION
